INTERFACE I_Frame

METHOD BlinkGreen : BOOL
VAR_INPUT
END_VAR
END_METHOD

PROPERTY ControlLeft : BOOL
GET
END_GET
END_PROPERTY

PROPERTY ControlRight : BOOL
GET
END_GET
END_PROPERTY

PROPERTY Door1 : BOOL
GET
END_GET
END_PROPERTY

PROPERTY Door2 : BOOL
GET
END_GET
END_PROPERTY

PROPERTY Door3 : BOOL
GET
END_GET
END_PROPERTY

PROPERTY GreenLight : BOOL
GET
END_GET
SET
END_SET
END_PROPERTY

END_INTERFACE

(* stored: Version 1.1.0.1, ProductVersion 3.1.4024.3
   Itf I_Frame: Id {8ca5ae50-405d-4929-9a0c-ad0b082ac295}
   Method BlinkGreen: Id {8b15ce8f-5bd2-48ba-8585-9a8d7f0efc10}
   Property ControlLeft: Id {e729e85a-80b6-4adc-8c85-644b890d8f09}
   Get Get: Id {a2373876-6400-4a3a-8ee9-c9c66b103bba}
   Property ControlRight: Id {c65635c4-bc85-4e2d-af33-c7c65dd1d083}
   Get Get: Id {d53d5e6b-04a4-47a2-8d8e-ad7cb1004761}
   Property Door1: Id {84c18a27-147d-4b73-9d3a-99ef2ade8586}
   Get Get: Id {dc3bd17a-6f81-4d0a-85af-8cab427feec1}
   Property Door2: Id {e872f46b-db9c-4669-89bc-4c41e1be477d}
   Get Get: Id {c90eea63-5803-49f8-9b39-9e2af68c6f2c}
   Property Door3: Id {6bd68c1e-2f1c-4655-940e-5ab0e7c0e7c6}
   Get Get: Id {eca6e6bc-3aaf-42f7-9f8c-8194ad116d89}
   Property GreenLight: Id {f606bc7a-66db-4f7f-a9d9-b435c4bda508}
   Get Get: Id {80539be2-cdb9-44cf-9ad7-85733403b2e6}
   Set Set: Id {459631e6-7b6f-4af0-8dcd-3b1bf86ed2d1} *)
